FUNCTION_BLOCK FB_MoveRel
VAR_INPUT
	targetDis		: LREAL;
	targetVel		: LREAL;
	execute			: BOOL := TRUE;
	
END_VAR

VAR_OUTPUT
	done 			: BOOL;
	moveRel			: Tc2_MC2.MC_MoveRelative;
END_VAR

VAR
	state		: INT := -10;
	power		: Tc2_MC2.MC_Power;
END_VAR

//Comment here
IF (NOT execute) THEN
	state := -10;
	moveRel	(Axis:= axis , Execute:= FALSE);
ELSE
	//Comment here
	power(
			Axis			:= axis , 
			Enable			:= TRUE , 
			Enable_Positive	:= TRUE , 
			Enable_Negative	:= TRUE , 
			BufferMode		:= Tc2_MC2.MC_BlendingNext
		);				
					
	CASE state OF 
		 
		-10:	//Comment here
				done := FALSE;
				IF (power.Status=TRUE AND power.Error=FALSE) THEN
					state := 0;
				END_IF
							
		0:		//Comment here
				moveRel(Axis:= axis , Execute:= FALSE);
				state := 10;			
				
		10:		//Comment here
				IF (moveRel.Done=FALSE) THEN
					moveRel(Axis:= axis, Execute:= TRUE, Distance:= targetDis, Velocity:=targetVel, BufferMode:= Tc2_MC2.MC_BlendingNext);
				ELSE 
					moveRel(Axis:= axis, Execute:= FALSE);
					state := 20;
				END_IF
				
		20: 	//Comment here
				done 	:= TRUE;
				execute := false;
				state	:= -10;	
	END_CASE
END_IF

END_FUNCTION_BLOCK

(* stored: Version 1.1.0.1, ProductVersion 3.1.0.25
   POU FB_MoveRel: Id {2907572c-55a5-4a40-a312-464a60ab1e0d} *)
